PROGRAM S03_LidChecking
VAR
	//工站
	station					: REFERENCE TO FB_Station:=fbstation[3];
	//气缸
	fbHOZAdjustCyl_1	:REFERENCE TO FB_Cylinder:=fbCylinder[12];	//	上层水平调整气缸1（小）
	fbHOZAdjustCyl_2	:REFERENCE TO FB_Cylinder:=fbCylinder[13];	//	上层水平调整气缸2（小）
	fbHOZAdjustCyl_3	:REFERENCE TO FB_Cylinder:=fbCylinder[14];	//	下层水平调整气缸1（小）
	fbHOZAdjustCyl_4	:REFERENCE TO FB_Cylinder:=fbCylinder[15];	//	下层水平调整气缸2（小）
	fbHOZAdjustCyl_5	:REFERENCE TO FB_Cylinder:=fbCylinder[16];	//	上层水平调整气缸1（大）
	fbHOZAdjustCyl_6	:REFERENCE TO FB_Cylinder:=fbCylinder[17];	//	上层水平调整气缸2（大）
	fbHOZAdjustCyl_7	:REFERENCE TO FB_Cylinder:=fbCylinder[18];	//	下层水平调整气缸1（大）
	fbHOZAdjustCyl_8	:REFERENCE TO FB_Cylinder:=fbCylinder[19];	//	下层水平调整气缸2（大）
	//伺服
	fbXAxisMove	 :REFERENCE TO FB_Axis:=fbAxis[6];	//	相机检测工位X轴伺服
	fbYAxisMove	 :REFERENCE TO FB_Axis:=fbAxis[7];	//	相机检测工位Y轴伺服
	fbZAxisMove	 :REFERENCE TO FB_Axis:=fbAxis[8];	//	相机检测工位Z轴伺服
	//相机

	
		//延时
		arTonDelay :ARRAY[1..20] OF TON;
	//返回值
		UdiReturnValue :ARRAY[1..20] OF UDINT;
	//本地过程数据
	arProcessDataStation : ARRAY [1..5] OF DUT_MainlineFixture;
	
	i,j: INT;
	
	// 循环计数
	bCounter: BYTE;
	// 临时变量
	_FirstCycle:ARRAY[1..10] OF BOOL;
	them: INT;
	// X轴伺服循环次数
	bXCounter: BYTE;
	// Y轴伺服循环次数
	bYCounter: BYTE;
	// 结束时循环次数
	bEndCounter: INT;
	//相机检测工位检测结果
	arCameraResult:ARRAY[1..5,1..4,1..12] OF INT;
	//过程记录
	tsModuleProcess:ARRAY[1..gc_ModuleProNo] OF DUT_Process;
	xClearModuleProcessDone:BOOL;
	bClearProcessStep	:BYTE;
END_VAR

A_Input();
Alarm();
Delay();
FlowAuto();
FlowInit();
General();
ILC();
TipAuto();
TipManual();
Z_Output();

ACTION A_Input:
//气缸
fbHOZAdjustCyl_1.xWP_Sensor	:=	IxS03HOZAdjustCyl_1WP	;
fbHOZAdjustCyl_1.xHP_Sensor	:=	IxS03HOZAdjustCyl_1HP	;
fbHOZAdjustCyl_2.xWP_Sensor	:=	IxS03HOZAdjustCyl_2WP	;
fbHOZAdjustCyl_2.xHP_Sensor	:=	IxS03HOZAdjustCyl_2HP	;
fbHOZAdjustCyl_3.xWP_Sensor	:=	IxS03HOZAdjustCyl_3WP	;
fbHOZAdjustCyl_3.xHP_Sensor	:=	IxS03HOZAdjustCyl_3HP	;
fbHOZAdjustCyl_4.xWP_Sensor	:=	IxS03HOZAdjustCyl_4WP	;
fbHOZAdjustCyl_4.xHP_Sensor	:=	IxS03HOZAdjustCyl_4HP	;
fbHOZAdjustCyl_5.xWP_Sensor	:=	IxS03HOZAdjustCyl_5WP	;
fbHOZAdjustCyl_5.xHP_Sensor	:=	IxS03HOZAdjustCyl_5HP	;
fbHOZAdjustCyl_6.xWP_Sensor	:=	IxS03HOZAdjustCyl_6WP	;
fbHOZAdjustCyl_6.xHP_Sensor	:=	IxS03HOZAdjustCyl_6HP	;
fbHOZAdjustCyl_7.xWP_Sensor	:=	IxS03HOZAdjustCyl_7WP	;
fbHOZAdjustCyl_7.xHP_Sensor	:=	IxS03HOZAdjustCyl_7HP	;
fbHOZAdjustCyl_8.xWP_Sensor	:=	IxS03HOZAdjustCyl_8WP	;
fbHOZAdjustCyl_8.xHP_Sensor	:=	IxS03HOZAdjustCyl_8HP	;
END_ACTION

ACTION Alarm:
station.adwAlarm[1].00	:=	station.xInitTimeout	;//	S03 初始化超时
station.adwAlarm[1].01	:=	fbHOZAdjustCyl_1.xHP_Off 	;//	S03上层水平调整气缸1(小)原点未到位
station.adwAlarm[1].02	:=	fbHOZAdjustCyl_1.xWP_Off 	;//	S03上层水平调整气缸1(小)动点未到位
station.adwAlarm[1].03	:=	fbHOZAdjustCyl_2.xHP_Off	;//	S03上层水平调整气缸2(小)原点未到位
station.adwAlarm[1].04	:=	fbHOZAdjustCyl_2.xWP_Off	;//	S03上层水平调整气缸2(小)动点未到位
station.adwAlarm[1].05	:=	fbHOZAdjustCyl_3.xHP_Off	;//	S03下层水平调整气缸1(小)原点未到位
station.adwAlarm[1].06	:=	fbHOZAdjustCyl_3.xWP_Off	;//	S03下层水平调整气缸1(小)动点未到位
station.adwAlarm[1].07	:=	fbHOZAdjustCyl_4.xHP_Off	;//	S03下层水平调整气缸2(小)原点未到位
station.adwAlarm[1].08	:=	fbHOZAdjustCyl_4.xWP_Off	;//	S03下层水平调整气缸2(小)动点未到位
station.adwAlarm[1].09	:=	fbHOZAdjustCyl_5.xHP_Off	;//	S03上层水平调整气缸1(大)原点未到位
station.adwAlarm[1].10	:=	fbHOZAdjustCyl_5.xWP_Off	;//	S03上层水平调整气缸1(大)动点未到位
station.adwAlarm[1].11	:=	fbHOZAdjustCyl_6.xHP_Off	;//	S03上层水平调整气缸2(大)原点未到位
station.adwAlarm[1].12	:=	fbHOZAdjustCyl_6.xWP_Off	;//	S03上层水平调整气缸2(大)动点未到位
station.adwAlarm[1].13	:=	fbHOZAdjustCyl_7.xHP_Off	;//	S03下层水平调整气缸1(大)原点未到位
station.adwAlarm[1].14	:=	fbHOZAdjustCyl_7.xWP_Off	;//	S03下层水平调整气缸1(大)动点未到位
station.adwAlarm[1].15	:=	fbHOZAdjustCyl_8.xHP_Off	;//	S03下层水平调整气缸2(大)原点未到位
station.adwAlarm[1].16	:=	fbHOZAdjustCyl_8.xWP_Off	;//	S03下层水平调整气缸2(大)动点未到位
station.adwAlarm[1].17	:=	fbXAxisMove.xError	;//	S03液位检测X轴伺服报错
station.adwAlarm[1].18	:=	fbXAxisMove.xNotPowerOn	;//	S03液位检测X轴伺服未使能
station.adwAlarm[1].19	:=	fbXAxisMove.xMoveTimeout	;//	S03液位检测X轴伺服移动超时
station.adwAlarm[1].20	:=	fbYAxisMove.xError	;//	S03液位检测Y轴伺服报错
station.adwAlarm[1].21	:=	fbYAxisMove.xNotPowerOn	;//	S03液位检测Y轴伺服未使能
station.adwAlarm[1].22	:=	fbYAxisMove.xMoveTimeout	;//	S03液位检测Y轴伺服移动超时
station.adwAlarm[1].23	:=	fbZAxisMove.xError	;//	S03液位检测Z轴伺服报错
station.adwAlarm[1].24	:=	fbZAxisMove.xNotPowerOn	;//	S03液位检测Z轴伺服未使能
station.adwAlarm[1].25	:=	fbZAxisMove.xMoveTimeout	;//	S03液位检测Z轴伺服移动超时
END_ACTION

ACTION Delay:
(*arTonDelay[01](IN:= , PT:=T#0.1S , Q=> , ET=> );*)//TipAuto使用
arTonDelay[02](IN:=  , PT:=T#1S , Q=> , ET=> );
arTonDelay[03](IN:=   , PT:=T#1S , Q=> , ET=> );
arTonDelay[04](IN:= , PT:=T#0.1S , Q=> , ET=> );
arTonDelay[05](IN:= , PT:=T#0.1S , Q=> , ET=> );
arTonDelay[06](IN:= , PT:=T#0.1S , Q=> , ET=> );
arTonDelay[07](IN:= , PT:=T#0.1S , Q=> , ET=> );
arTonDelay[08](IN:= , PT:=T#0.1S , Q=> , ET=> );
arTonDelay[09](IN:= , PT:=T#0.1S , Q=> , ET=> );
END_ACTION

ACTION FlowAuto:

//-----------------------------------------初始化是否完成判断----------------------------------------------
IF NOT station.xInitDone 
THEN
 	station.iStepAuto:=0;
 	station.xDone:=FALSE;
	station.xRunningOffProhibit := FALSE ;//运行中信号Off禁止
ELSIF station.xRunning  OR (tsModuleProcess[bXCounter+1].xProcessStarted AND NOT tsModuleProcess[bXCounter+1].xProcessCompleted)
THEN
//-----------------------------------------动作步骤--------------------------------------------------------
CASE station.iStepAuto OF	  
	0: //----Home Step，等待启动----
		IF station.xDisabled 
			AND station.xCanRun 
			AND NOT fbMachine[1].xStopped 
			AND NOT station.xSingleRunning 
		THEN
			station.xDone:=TRUE;
		END_IF
		
		IF  station.xSingleRunning 
			OR station.xCanRun 
			AND NOT station.xDone 
			AND NOT station.xDisabled 
			AND NOT fbMachine[1].xStopped
		THEN
			station.xCycleEnable:=TRUE;
			station.xDone:= FALSE;  
			station.iStepAuto:= 5;
		END_IF		
	 5://复位数据
			IF  station.xSingleRunning THEN
				 FOR i:=1 TO gc_ModuleProNo BY 1 DO
						 MEMSET(ADR(tsModuleProcess[i]),0,SIZEOF(tsModuleProcess[i]));
				 END_FOR
			END_IF	
			station.iStepAuto:= 10;
	 10: //判断产品是否到该工位
		IF  station.xSingleRunning THEN
			station.iStepAuto:= 11;
		ELSIF fbMachine[1].xTryRun THEN
			IF NOT _FirstCycle[6] THEN
					bCounter:=1;
					bEndCounter:=0;
				_FirstCycle[6]:=TRUE;
			END_IF
			station.iStepAuto:= 11;
		ELSE
			IF   	 NOT  arMainlineFixtureData[arCurFixtureNumStation[5]].xMaterialOnOff AND
					 NOT arMainlineFixtureData[arCurFixtureNumStation[6]].xMaterialOnOff  AND 
					 NOT arMainlineFixtureData[arCurFixtureNumStation[7]].xMaterialOnOff AND 
					NOT	arMainlineFixtureData[arCurFixtureNumStation[8]].xMaterialOnOff AND
					NOT arMainlineFixtureData[arCurFixtureNumStation[9]].xMaterialOnOff  THEN
							bCounter:=0;
							bEndCounter :=0;
							_FirstCycle[1]:=FALSE;
							_FirstCycle[2]:=FALSE;
							_FirstCycle[6]:=FALSE;
							station.iStepAuto:= 999;
						
			ELSIF	 arMainlineFixtureData[arCurFixtureNumStation[5]].xMaterialOnOff AND    
				    arMainlineFixtureData[arCurFixtureNumStation[6]].xMaterialOnOff (* AND 
				NOT arMainlineFixtureData[arCurFixtureNumStation[7]].xMaterialOnOff AND 
				NOT	arMainlineFixtureData[arCurFixtureNumStation[8]].xMaterialOnOff AND
				NOT arMainlineFixtureData[arCurFixtureNumStation[9]].xMaterialOnOff*)  THEN
					IF  NOT _FirstCycle[1] THEN
							bCounter:=1;
							bEndCounter :=0;
							_FirstCycle[1]:=TRUE;
					END_IF
					station.iStepAuto:= 11;
			ELSIF   NOT arMainlineFixtureData[arCurFixtureNumStation[5]].xMaterialOnOff AND    
				    NOT arMainlineFixtureData[arCurFixtureNumStation[6]].xMaterialOnOff  AND 
						arMainlineFixtureData[arCurFixtureNumStation[7]].xMaterialOnOff AND 
						arMainlineFixtureData[arCurFixtureNumStation[8]].xMaterialOnOff AND
						arMainlineFixtureData[arCurFixtureNumStation[9]].xMaterialOnOff  THEN
					IF  NOT _FirstCycle[2] THEN
							bEndCounter:=1;
							bCounter:=0;
							_FirstCycle[2]:=TRUE;
					END_IF
					station.iStepAuto:= 11;
			END_IF
		END_IF
	11://手动NOK按钮
			IF   arManualNOKHmiButton[3]  AND NOT station.xSingleRunning THEN
				station.iStepAuto:= 280;
			ELSE	
				station.iStepAuto:= 20;
			END_IF
			
	20:////Restore_after_Estop_Process1 上载数据流程
			IF   station.xSingleRunning OR  fbMachine[1].xTryRun THEN
				    station.iStepAuto :=40;
			ELSIF tsModuleProcess[1].xProcessNotStarted AND NOT  tsModuleProcess[1].xProcessStarted THEN
					station.iStepAuto :=21; (*process not started*)
			ELSIF  tsModuleProcess[1].xProcessStarted AND NOT  tsModuleProcess[1].xProcessCompleted THEN
				 station.iStepAuto := 21;(*process started*)
			ELSIF  tsModuleProcess[1].xProcessCompleted AND NOT tsModuleProcess[1].xQDataCompleted  THEN
					station.iStepAuto := 40 ;(*process completed*)
			ELSIF tsModuleProcess[1].xQDataCompleted THEN
					station.iStepAuto :=40;(*Qdata completed *)
			ELSE
					station.iStepAuto :=21; 
			END_IF	
	21://
				tsModuleProcess[1].xProcessNotStarted:=TRUE;
				station.iStepAuto:= 30;
	30://上载产品数据
			tsModuleProcess[1].xProcessStarted	:=TRUE;
			IF  bCounter =1 OR bCounter =2 OR bCounter=3 THEN
				MEMCPY(ADR(arProcessDataStation[1]),ADR(arMainlineFixtureData[arCurFixtureNumStation[5]]),SIZEOF(arMainlineFixtureData[arCurFixtureNumStation[5]]));
				MEMCPY(ADR(arProcessDataStation[2]),ADR(arMainlineFixtureData[arCurFixtureNumStation[6]]),SIZEOF(arMainlineFixtureData[arCurFixtureNumStation[6]]))	;
			END_IF
			IF bCounter =2 OR bCounter =3 OR bEndCounter =1 THEN
				MEMCPY(ADR(arProcessDataStation[3]),ADR(arMainlineFixtureData[arCurFixtureNumStation[7]]),SIZEOF(arMainlineFixtureData[arCurFixtureNumStation[7]]));
				MEMCPY(ADR(arProcessDataStation[4]),ADR(arMainlineFixtureData[arCurFixtureNumStation[8]]),SIZEOF(arMainlineFixtureData[arCurFixtureNumStation[8]]))	;
			END_IF
			IF bCounter =3 OR bEndCounter =2 THEN
				MEMCPY(ADR(arProcessDataStation[5]),ADR(arMainlineFixtureData[arCurFixtureNumStation[9]]),SIZEOF(arMainlineFixtureData[arCurFixtureNumStation[9]]))	;
			END_IF
			tsModuleProcess[1].xProcessCompleted:=TRUE;
			station.iStepAuto:= 40;
	/////产品流程开始	
		40://设定X轴循环为1，总次数2
				 bXCounter:=1;
				station.iStepAuto:= 50;		
		50:////Restore_after_Estop_Process2/3 X轴位置1/2拍照流程
			 IF  station.xSingleRunning OR fbMachine[1].xTryRun THEN
					 station.iStepAuto :=70; 
			 ELSIF tsModuleProcess[bXCounter+1].xProcessNotStarted AND NOT  tsModuleProcess[bXCounter+1].xProcessStarted THEN
					 station.iStepAuto :=70; (*process not started*)
			 ELSIF  tsModuleProcess[bXCounter+1].xProcessStarted AND NOT  tsModuleProcess[bXCounter+1].xProcessCompleted THEN
					station.iStepAuto := 70;(*process started*)
			 ELSIF  tsModuleProcess[bXCounter+1].xProcessCompleted AND NOT tsModuleProcess[bXCounter+1].xQDataCompleted  THEN
					 station.iStepAuto :=200;(*process completed*)
			 ELSIF tsModuleProcess[bXCounter+1].xQDataCompleted THEN
					 station.iStepAuto :=200;(*Qdata completed *)
			 ELSE
					 station.iStepAuto :=70; 
			 END_IF	
		70://流程未开始
				tsModuleProcess[bXCounter+1].xProcessNotStarted :=TRUE;
				station.iStepAuto :=80; 
		80://水平调整气缸伸出		
			IF   bCounter =1 THEN
					IF  iBoxChoose =1 THEN
						(*上层水平调整气缸*)
						fbHOZAdjustCyl_1.xAuto :=TRUE;
						fbHOZAdjustCyl_2.xAuto :=TRUE;
						IF  fbHOZAdjustCyl_1.xWP_Delay AND fbHOZAdjustCyl_2.xWP_Delay  THEN
								station.iStepAuto:= 90;
						END_IF
					ELSIF  iBoxChoose= 2 THEN
						(*下层水平调整气缸*)
						fbHOZAdjustCyl_3.xAuto :=TRUE;
						fbHOZAdjustCyl_4.xAuto :=TRUE;
						IF  fbHOZAdjustCyl_3.xWP_Delay AND fbHOZAdjustCyl_4.xWP_Delay  THEN
								station.iStepAuto:= 90;
						END_IF
					END_IF
			ELSIF  bCounter =2 OR  bCounter =3 OR bEndCounter =1 OR bEndCounter =2 THEN
					IF  iBoxChoose =1 THEN
						(*上层水平调整气缸*)
						fbHOZAdjustCyl_5.xAuto :=TRUE;
						fbHOZAdjustCyl_6.xAuto :=TRUE;
						IF  fbHOZAdjustCyl_5.xWP_Delay AND fbHOZAdjustCyl_6.xWP_Delay  THEN
								station.iStepAuto:= 90;
						END_IF
					ELSIF  iBoxChoose= 2 THEN
						(*下层水平调整气缸*)
						fbHOZAdjustCyl_7.xAuto :=TRUE;
						fbHOZAdjustCyl_8.xAuto :=TRUE;
						IF  fbHOZAdjustCyl_7.xWP_Delay AND fbHOZAdjustCyl_8.xWP_Delay  THEN
								station.iStepAuto:= 90;
						END_IF
					END_IF
			END_IF
		90://Z轴下降
			fbZAxisMove.xMoveAuto[2]:=TRUE;
			IF  fbXAxisMove.xMoveInPos[2] THEN
				station.iStepAuto:= 95;
			END_IF			 
		95://X轴移动到拍照位置1/2
				fbXAxisMove.xMoveAuto[bXCounter+1]:=TRUE;
				IF  fbXAxisMove.xMoveInPos[bXCounter+1] THEN
					station.iStepAuto:= 100;
				END_IF
		100://设定Y轴循环开始 总次数为3
				 bYCounter:=1;
				station.iStepAuto:= 110;	
		110://Y轴移动到位置1/2/3	
				fbYAxisMove.xMoveAuto[bYCounter+1]:=TRUE;
				IF  fbYAxisMove.xMoveInPos[bYCounter+1] THEN
					station.iStepAuto:= 120;
				END_IF
		120://屏蔽拍照
			IF axBypassSignal[3] OR  fbMachine[1].xTryRun THEN
 					station.iStepAuto:= 150;	
			ELSE
					station.iStepAuto:= 140;		
			END_IF
		140://触发拍照
			(*开始循环*)
			tsModuleProcess[bXCounter+1].xProcessStarted :=TRUE;
			IF   bCounter =1  (*17.18位置有产品*)  THEN
					IF  bXCounter =1 THEN
							FOR i:=2 TO  9 BY 1 DO
								fbCamera[i].xlTrigger:=TRUE;
							END_FOR
					ELSIF bXCounter =2 THEN
							FOR i:=2 TO  5 BY 1 DO
								fbCamera[i].xlTrigger:=TRUE;
							END_FOR
					END_IF
			ELSIF  bCounter=2  THEN
					IF  bXCounter =1 THEN
								FOR i:=2 TO 17 BY 1 DO
									fbCamera[i].xlTrigger:=TRUE;
								END_FOR
					ELSIF   bXCounter =2 THEN
								FOR i:=2 TO 13 BY 1 DO
									fbCamera[i].xlTrigger:=TRUE;
								END_FOR	
					END_IF
			ELSIF   bCounter=3 THEN
					FOR i:=2 TO 17 BY 1 DO
						fbCamera[i].xlTrigger:=TRUE;
					END_FOR
			END_IF
			(*结束循环*)
			IF   bEndCounter =1 (*17.18位置无产品*)  THEN
					IF  bXCounter =1 THEN
								FOR i:=6 TO  17 BY 1 DO
									fbCamera[i].xlTrigger:=TRUE;
								END_FOR
					ELSIF bXCounter =2 THEN
								FOR i:=2 TO  17 BY 1 DO
									fbCamera[i].xlTrigger:=TRUE;
								END_FOR
					END_IF
			ELSIF  bEndCounter =2 THEN
					IF bXCounter =2 THEN
							FOR i:=14 TO  17 BY 1 DO
									fbCamera[i].xlTrigger:=TRUE;
							END_FOR	
					END_IF
			END_IF
			FOR i:=2 TO 17 BY 1 DO
				IF  fbCamera[i].xQBusy  THEN
					fbCamera[i].xlTrigger:=FALSE;
					station.iStepAuto:=150;
				END_IF
			END_FOR
		150://检查相机完成信号并储存
		(*开始循环*)
			 IF   bCounter =1 (*17.18位置有产品*)  THEN	
				  	IF  bXCounter =1 THEN
							IF   axBypassSignal[3] OR  fbMachine[1].xTryRun THEN
								
											arCameraResult[1,3,bYCounter]:=1;	
											arCameraResult[1,3,6+bYCounter]:=1;	
											arCameraResult[1,1,3+bYCounter]:=1;
											arCameraResult[1,1,9+bYCounter]:=1;
											arCameraResult[2,4,bYCounter]:=1;
											arCameraResult[2,4,6+bYCounter]:=1;
											arCameraResult[2,2,3+bYCounter]:=1;
											arCameraResult[2,2,9+bYCounter]:=1;	
											station.iStepAuto:=160;
							ELSE
								FOR i:=1 TO  8 BY 1 DO
										IF  fbCamera[i].xQBusy THEN	
												EXIT;
										ELSE
												IF  i =1 THEN
													arCameraResult[1,3,bYCounter]:=sCamera_To_Plc.iS03Result[i];	
												ELSIF i =2 THEN
													arCameraResult[1,3,6+bYCounter]:=sCamera_To_Plc.iS03Result[i];	
												ELSIF i =3 THEN
													arCameraResult[1,1,3+bYCounter]:=sCamera_To_Plc.iS03Result[i];
												ELSIF i =4 THEN
													arCameraResult[1,1,9+bYCounter]:=sCamera_To_Plc.iS03Result[i];
												ELSIF i =5 THEN
													arCameraResult[2,4,bYCounter]:=sCamera_To_Plc.iS03Result[i];
												ELSIF i =6 THEN
													arCameraResult[2,4,6+bYCounter]:=sCamera_To_Plc.iS03Result[i];
												ELSIF i =7 THEN
													arCameraResult[2,2,3+bYCounter]:=sCamera_To_Plc.iS03Result[i];
												ELSIF i =8 THEN
													arCameraResult[2,2,9+bYCounter]:=sCamera_To_Plc.iS03Result[i];	
												END_IF	
										END_IF
										IF   i =8 THEN
											station.iStepAuto:=160;
										END_IF
								END_FOR
							END_IF
				
				 	ELSIF   bXCounter =2 THEN
							IF   axBypassSignal[3] OR  fbMachine[1].xTryRun THEN
											arCameraResult[2,3,bYCounter]:=1;	
											arCameraResult[2,3,6+bYCounter]:=1;	
											arCameraResult[2,1,3+bYCounter]:=1;
											arCameraResult[2,1,9+bYCounter]:=1;
											station.iStepAuto:=160;
							ELSE
								FOR i:=1 TO 4 BY 1	DO
										IF  fbCamera[i].xQBusy THEN	
											EXIT;
										ELSE
											IF  i =1 THEN
												arCameraResult[2,3,bYCounter]:=sCamera_To_Plc.iS03Result[i];	
											ELSIF i =2 THEN
												arCameraResult[2,3,6+bYCounter]:=sCamera_To_Plc.iS03Result[i];	
											ELSIF i =3 THEN
												arCameraResult[2,1,3+bYCounter]:=sCamera_To_Plc.iS03Result[i];
											ELSIF i =4 THEN
												arCameraResult[2,1,9+bYCounter]:=sCamera_To_Plc.iS03Result[i];
											END_IF
										END_IF	
										IF   i =8 THEN
											station.iStepAuto:=160;
										END_IF
								END_FOR
							END_IF
							
					END_IF		
			ELSIF  bCounter=2 THEN
					IF bXCounter =1 THEN
							IF   axBypassSignal[3] OR  fbMachine[1].xTryRun THEN
									
												arCameraResult[1,3,bYCounter]:=1;	
												arCameraResult[1,3,6+bYCounter]:=1;	
												arCameraResult[1,1,3+bYCounter]:=1;
												arCameraResult[1,1,9+bYCounter]:=1;
												arCameraResult[2,4,bYCounter]:=1;
												arCameraResult[2,4,6+bYCounter]:=1;
												arCameraResult[2,2,3+bYCounter]:=1;
												arCameraResult[2,2,9+bYCounter]:=1;	
												arCameraResult[3,3,3+bYCounter]:=1;	
												arCameraResult[3,3,9+bYCounter]:=1;	
												arCameraResult[3,1,bYCounter]:= 1;
												arCameraResult[3,1,6+bYCounter]:=1;
												arCameraResult[4,4,3+bYCounter]:=1;
												arCameraResult[4,4,9+bYCounter]:=1;
												arCameraResult[4,2,3+bYCounter]:=1;
												arCameraResult[4,2,6+bYCounter]:=1;	
												station.iStepAuto:=160;
							ELSE
								FOR i:=1 TO  16 BY 1 DO
									IF  fbCamera[i].xQBusy THEN	
											EXIT;
									ELSE
											IF  i =1 THEN
												arCameraResult[1,3,bYCounter]:=sCamera_To_Plc.iS03Result[i];	
											ELSIF i =2 THEN
												arCameraResult[1,3,6+bYCounter]:=sCamera_To_Plc.iS03Result[i];	
											ELSIF i =3 THEN
												arCameraResult[1,1,3+bYCounter]:=sCamera_To_Plc.iS03Result[i];
											ELSIF i =4 THEN
												arCameraResult[1,1,9+bYCounter]:=sCamera_To_Plc.iS03Result[i];
											ELSIF i =5 THEN
												arCameraResult[2,4,bYCounter]:=sCamera_To_Plc.iS03Result[i];
											ELSIF i =6 THEN
												arCameraResult[2,4,6+bYCounter]:=sCamera_To_Plc.iS03Result[i];
											ELSIF i =7 THEN
												arCameraResult[2,2,3+bYCounter]:=sCamera_To_Plc.iS03Result[i];
											ELSIF i =8 THEN
												arCameraResult[2,2,9+bYCounter]:=sCamera_To_Plc.iS03Result[i];	
											ELSIF i =9 THEN
												arCameraResult[3,3,3+bYCounter]:=sCamera_To_Plc.iS03Result[i];	
											ELSIF i =10 THEN
												arCameraResult[3,3,9+bYCounter]:=sCamera_To_Plc.iS03Result[i];	
											ELSIF i =11 THEN
												arCameraResult[3,1,bYCounter]:=sCamera_To_Plc.iS03Result[i];
											ELSIF i =12 THEN
												arCameraResult[3,1,6+bYCounter]:=sCamera_To_Plc.iS03Result[i];
											ELSIF i =13 THEN
												arCameraResult[4,4,3+bYCounter]:=sCamera_To_Plc.iS03Result[i];
											ELSIF i =14 THEN
												arCameraResult[4,4,9+bYCounter]:=sCamera_To_Plc.iS03Result[i];
											ELSIF i =15 THEN
												arCameraResult[4,2,3+bYCounter]:=sCamera_To_Plc.iS03Result[i];
											ELSIF i =16 THEN
												arCameraResult[4,2,6+bYCounter]:=sCamera_To_Plc.iS03Result[i];	
											END_IF	
									END_IF	
									IF   i =16 THEN
											station.iStepAuto:=160;
									END_IF
								END_FOR	
							END_IF
							
					ELSIF bXCounter =2 THEN
							IF   axBypassSignal[3] OR  fbMachine[1].xTryRun THEN
											arCameraResult[2,3,bYCounter]:=1;	
											arCameraResult[2,3,6+bYCounter]:=1;	
											arCameraResult[2,1,3+bYCounter]:=1;
											arCameraResult[2,1,9+bYCounter]:=1;
											arCameraResult[3,4,bYCounter]:=1;
											arCameraResult[3,4,6+bYCounter]:=1;
											arCameraResult[3,2,3+bYCounter]:=1;
											arCameraResult[3,2,9+bYCounter]:=1;	
											arCameraResult[4,3,3+bYCounter]:=1;	
											arCameraResult[4,3,9+bYCounter]:=1;	
											arCameraResult[4,1,bYCounter]:=1;
											arCameraResult[4,1,6+bYCounter]:=1;
											station.iStepAuto:=160;
							ELSE
								FOR i:=1 TO  12 BY 1 DO
									IF  fbCamera[i].xQBusy THEN	
											EXIT;
									ELSE
											IF  i =1 THEN
												arCameraResult[2,3,bYCounter]:=sCamera_To_Plc.iS03Result[i];	
											ELSIF i =2 THEN       
												arCameraResult[2,3,6+bYCounter]:=sCamera_To_Plc.iS03Result[i];	
											ELSIF i =3 THEN      
												arCameraResult[2,1,3+bYCounter]:=sCamera_To_Plc.iS03Result[i];
											ELSIF i =4 THEN      
												arCameraResult[2,1,9+bYCounter]:=sCamera_To_Plc.iS03Result[i];
											ELSIF i =5 THEN      
												arCameraResult[3,4,bYCounter]:=sCamera_To_Plc.iS03Result[i];
											ELSIF i =6 THEN     
												arCameraResult[3,4,6+bYCounter]:=sCamera_To_Plc.iS03Result[i];
											ELSIF i =7 THEN      
												arCameraResult[3,2,3+bYCounter]:=sCamera_To_Plc.iS03Result[i];
											ELSIF i =8 THEN      
												arCameraResult[3,2,9+bYCounter]:=sCamera_To_Plc.iS03Result[i];	
											ELSIF i =9 THEN      
												arCameraResult[4,3,3+bYCounter]:=sCamera_To_Plc.iS03Result[i];	
											ELSIF i =10 THEN     
												arCameraResult[4,3,9+bYCounter]:=sCamera_To_Plc.iS03Result[i];	
											ELSIF i =11 THEN      
												arCameraResult[4,1,bYCounter]:=sCamera_To_Plc.iS03Result[i];
											ELSIF i =12 THEN      
												arCameraResult[4,1,6+bYCounter]:=sCamera_To_Plc.iS03Result[i];
											END_IF	
									END_IF
									IF   i =12 THEN
										station.iStepAuto:=160;
									END_IF	
								END_FOR	
							END_IF
					END_IF
				
			ELSIF  bCounter =3 THEN
					IF bXCounter =1 THEN
							IF   axBypassSignal[3] OR  fbMachine[1].xTryRun THEN
								
											arCameraResult[1,3,bYCounter]:=	1;	
											arCameraResult[1,3,6+bYCounter]:=1;	
											arCameraResult[1,1,3+bYCounter]:=1;
											arCameraResult[1,1,9+bYCounter]:=1;
											arCameraResult[2,4,bYCounter]:=1;
											arCameraResult[2,4,6+bYCounter]:=1;
											arCameraResult[2,2,3+bYCounter]:=1;
											arCameraResult[2,2,9+bYCounter]:=1;	
											arCameraResult[3,3,3+bYCounter]:=1;	
											arCameraResult[3,3,9+bYCounter]:=1;	
											arCameraResult[3,1,bYCounter]:=1;
											arCameraResult[3,1,6+bYCounter]:=1;
											arCameraResult[4,4,3+bYCounter]:=1;
											arCameraResult[4,4,9+bYCounter]:=1;
											arCameraResult[4,2,3+bYCounter]:=1;
											arCameraResult[4,2,6+bYCounter]:=1;	
											station.iStepAuto:=160;
							ELSE
								FOR i:=1 TO  16 BY 1 DO
										IF  fbCamera[i].xQBusy THEN	
												EXIT;
										ELSE
												IF  i =1 THEN
													arCameraResult[1,3,bYCounter]:=sCamera_To_Plc.iS03Result[i];	
												ELSIF i =2 THEN   
													arCameraResult[1,3,6+bYCounter]:=sCamera_To_Plc.iS03Result[i];	
												ELSIF i =3 THEN    
													arCameraResult[1,1,3+bYCounter]:=sCamera_To_Plc.iS03Result[i];
												ELSIF i =4 THEN    
													arCameraResult[1,1,9+bYCounter]:=sCamera_To_Plc.iS03Result[i];
												ELSIF i =5 THEN     
													arCameraResult[2,4,bYCounter]:=sCamera_To_Plc.iS03Result[i];
												ELSIF i =6 THEN    
													arCameraResult[2,4,6+bYCounter]:=sCamera_To_Plc.iS03Result[i];
												ELSIF i =7 THEN     
													arCameraResult[2,2,3+bYCounter]:=sCamera_To_Plc.iS03Result[i];
												ELSIF i =8 THEN     
													arCameraResult[2,2,9+bYCounter]:=sCamera_To_Plc.iS03Result[i];	
												ELSIF i =9 THEN     
													arCameraResult[3,3,3+bYCounter]:=sCamera_To_Plc.iS03Result[i];	
												ELSIF i =10 THEN    
													arCameraResult[3,3,9+bYCounter]:=sCamera_To_Plc.iS03Result[i];	
												ELSIF i =11 THEN    
													arCameraResult[3,1,bYCounter]:=sCamera_To_Plc.iS03Result[i];
												ELSIF i =12 THEN    
													arCameraResult[3,1,6+bYCounter]:=sCamera_To_Plc.iS03Result[i];
												ELSIF i =13 THEN    
													arCameraResult[4,4,3+bYCounter]:=sCamera_To_Plc.iS03Result[i];
												ELSIF i =14 THEN    
													arCameraResult[4,4,9+bYCounter]:=sCamera_To_Plc.iS03Result[i];
												ELSIF i =15 THEN    
													arCameraResult[4,2,3+bYCounter]:=sCamera_To_Plc.iS03Result[i];
												ELSIF i =16 THEN   
													arCameraResult[4,2,6+bYCounter]:=sCamera_To_Plc.iS03Result[i];	
												END_IF	
										END_IF	
										IF  i =16 THEN 
											station.iStepAuto:=160;
										END_IF
								END_FOR	
							END_IF
					ELSIF bXCounter =2 THEN
							IF   axBypassSignal[3] OR  fbMachine[1].xTryRun THEN
								
												arCameraResult[2,3,bYCounter]:=1;	
											arCameraResult[2,3,6+bYCounter]:=1;	
											arCameraResult[2,1,3+bYCounter]:=1;
											arCameraResult[2,1,9+bYCounter]:=1;
											arCameraResult[3,4,bYCounter]:=1;
											arCameraResult[3,4,6+bYCounter]:=1;
											arCameraResult[3,2,3+bYCounter]:=1;
											arCameraResult[3,2,9+bYCounter]:=1;	
											arCameraResult[4,3,3+bYCounter]:=1;	
											arCameraResult[4,3,9+bYCounter]:=1;	
											arCameraResult[4,1,bYCounter]:=1;
											arCameraResult[4,1,6+bYCounter]:=1;
											arCameraResult[5,4,3+bYCounter]:=1;
											arCameraResult[5,4,9+bYCounter]:=1;
											arCameraResult[5,2,3+bYCounter]:=1;
											arCameraResult[5,2,6+bYCounter]:=1;	
											station.iStepAuto:=160;
							ELSE
								FOR i:=1 TO  12 BY 1 DO
									IF fbCamera[i].xQBusy THEN	
											EXIT;
									ELSE
											IF  i =1 THEN
												arCameraResult[2,3,bYCounter]:=sCamera_To_Plc.iS03Result[i];	
											ELSIF i =2 THEN   
												arCameraResult[2,3,6+bYCounter]:=sCamera_To_Plc.iS03Result[i];	
											ELSIF i =3 THEN    
												arCameraResult[2,1,3+bYCounter]:=sCamera_To_Plc.iS03Result[i];
											ELSIF i =4 THEN     
												arCameraResult[2,1,9+bYCounter]:=sCamera_To_Plc.iS03Result[i];
											ELSIF i =5 THEN     
												arCameraResult[3,4,bYCounter]:=sCamera_To_Plc.iS03Result[i];
											ELSIF i =6 THEN    
												arCameraResult[3,4,6+bYCounter]:=sCamera_To_Plc.iS03Result[i];
											ELSIF i =7 THEN   
												arCameraResult[3,2,3+bYCounter]:=sCamera_To_Plc.iS03Result[i];
											ELSIF i =8 THEN     
												arCameraResult[3,2,9+bYCounter]:=sCamera_To_Plc.iS03Result[i];	
											ELSIF i =9 THEN    
												arCameraResult[4,3,3+bYCounter]:=sCamera_To_Plc.iS03Result[i];	
											ELSIF i =10 THEN    
												arCameraResult[4,3,9+bYCounter]:=sCamera_To_Plc.iS03Result[i];	
											ELSIF i =11 THEN    
												arCameraResult[4,1,bYCounter]:=sCamera_To_Plc.iS03Result[i];
											ELSIF i =12 THEN    
												arCameraResult[4,1,6+bYCounter]:=sCamera_To_Plc.iS03Result[i];
											ELSIF i =13 THEN   
												arCameraResult[5,4,3+bYCounter]:=sCamera_To_Plc.iS03Result[i];
											ELSIF i =14 THEN    
												arCameraResult[5,4,9+bYCounter]:=sCamera_To_Plc.iS03Result[i];
											ELSIF i =15 THEN    
												arCameraResult[5,2,3+bYCounter]:=sCamera_To_Plc.iS03Result[i];
											ELSIF i =16 THEN   
												arCameraResult[5,2,6+bYCounter]:=sCamera_To_Plc.iS03Result[i];	
											END_IF	
									END_IF
									IF  i =12 THEN
										station.iStepAuto:=160;	
									END_IF
								END_FOR	
							END_IF
					END_IF
			END_IF
			
		(*结束循环*)
			 IF   bEndCounter =1 (*17.18位置无产品*)  THEN	
				  	IF  bXCounter =1 THEN
							IF   axBypassSignal[3] OR  fbMachine[1].xTryRun THEN
											arCameraResult[3,3,3+bYCounter]:=1;
											arCameraResult[3,3,9+bYCounter]:=1;
											arCameraResult[3,1,bYCounter]:=1;
											arCameraResult[3,1,3+bYCounter]:=1;                 
											arCameraResult[4,4,3+bYCounter]:=1;	
											arCameraResult[4,4,9+bYCounter]:=1;
											arCameraResult[4,2,bYCounter]:=1;
											arCameraResult[4,2,6+bYCounter]:=1;
											station.iStepAuto:=160;
							ELSE
								FOR i:=9 TO  16 BY 1 DO
									IF  fbCamera[i].xQBusy THEN	
											EXIT;
									ELSE
											IF i =9 THEN
												arCameraResult[3,3,3+bYCounter]:=sCamera_To_Plc.iS03Result[i];
											ELSIF i =10 THEN   
												arCameraResult[3,3,9+bYCounter]:=sCamera_To_Plc.iS03Result[i];
											ELSIF i =11 THEN   
												arCameraResult[3,1,bYCounter]:=sCamera_To_Plc.iS03Result[i];
											ELSIF i =12 THEN    
												arCameraResult[3,1,3+bYCounter]:=sCamera_To_Plc.iS03Result[i];                 
											ELSIF i =13 THEN   
												arCameraResult[4,4,3+bYCounter]:=sCamera_To_Plc.iS03Result[i];	
											ELSIF i =14 THEN    
												arCameraResult[4,4,9+bYCounter]:=sCamera_To_Plc.iS03Result[i];
											ELSIF i =15 THEN    
												arCameraResult[4,2,bYCounter]:=sCamera_To_Plc.iS03Result[i];
											ELSIF i =16 THEN   
												arCameraResult[4,2,6+bYCounter]:=sCamera_To_Plc.iS03Result[i];
											END_IF
									END_IF	
									IF  i =16 THEN
											station.iStepAuto:=160;	
									END_IF
								END_FOR	
							END_IF
							
				 	ELSIF   bXCounter =2 THEN
							IF   axBypassSignal[3] OR  fbMachine[1].xTryRun THEN
							
											arCameraResult[3,4,bYCounter]:=1;	
											arCameraResult[3,4,6+bYCounter]:=1;	
											arCameraResult[3,2,3+bYCounter]:=1;
											arCameraResult[3,2,9+bYCounter]:=1;
											arCameraResult[4,3,3+bYCounter]:=1;	
											arCameraResult[4,3,8+bYCounter]:=1;	
											arCameraResult[4,1,bYCounter]:=1;
											arCameraResult[4,1,6+bYCounter]:=1;		
											arCameraResult[5,4,3+bYCounter]:=1;	
											arCameraResult[5,4,9+bYCounter]:=1;	
											arCameraResult[5,2,bYCounter]:=1;
											arCameraResult[5,2,6+bYCounter]:=1;
											station.iStepAuto:=160;
							ELSE
								FOR i:=5 TO 16 BY 1	DO
										IF  fbCamera[i].xQBusy THEN	
											EXIT;
										ELSE
											IF  i =5 THEN
												arCameraResult[3,4,bYCounter]:=sCamera_To_Plc.iS03Result[i];	
											ELSIF i =6 THEN    
												arCameraResult[3,4,6+bYCounter]:=sCamera_To_Plc.iS03Result[i];	
											ELSIF i =7 THEN    
												arCameraResult[3,2,3+bYCounter]:=sCamera_To_Plc.iS03Result[i];
											ELSIF i =8 THEN    
												arCameraResult[3,2,9+bYCounter]:=sCamera_To_Plc.iS03Result[i];
											ELSIF  i =9 THEN    
												arCameraResult[4,3,3+bYCounter]:=sCamera_To_Plc.iS03Result[i];	
											ELSIF i =10 THEN    
												arCameraResult[4,3,8+bYCounter]:=sCamera_To_Plc.iS03Result[i];	
											ELSIF i =11 THEN    
												arCameraResult[4,1,bYCounter]:=sCamera_To_Plc.iS03Result[i];
											ELSIF i =12 THEN  
												arCameraResult[4,1,6+bYCounter]:=sCamera_To_Plc.iS03Result[i];		
											ELSIF  i =13 THEN 
												arCameraResult[5,4,3+bYCounter]:=sCamera_To_Plc.iS03Result[i];	
											ELSIF i =14 THEN   
												arCameraResult[5,4,9+bYCounter]:=sCamera_To_Plc.iS03Result[i];	
											ELSIF i =15 THEN   
												arCameraResult[5,2,bYCounter]:=sCamera_To_Plc.iS03Result[i];
											ELSIF i =16 THEN  
												arCameraResult[5,2,6+bYCounter]:=sCamera_To_Plc.iS03Result[i];
											END_IF
										END_IF
										IF i =16 THEN
											station.iStepAuto:=160;
										END_IF
								END_FOR
							END_IF
							
						END_IF		
			ELSIF  bEndCounter=2 THEN
					IF bXCounter =2 THEN
							IF   axBypassSignal[3] OR  fbMachine[1].xTryRun THEN
								
												arCameraResult[5,4,3+bYCounter]:=1;	
												arCameraResult[5,4,9+bYCounter]:=1;	
												arCameraResult[5,4,bYCounter]:=1;
												arCameraResult[5,4,6+bYCounter]:=1;
												station.iStepAuto:=160;
							ELSE
								FOR i:=13 TO  16 BY 1 DO
									IF  fbCamera[i].xQBusy THEN	
											EXIT;
									ELSE
											IF  i =13 THEN
												arCameraResult[5,4,3+bYCounter]:=sCamera_To_Plc.iS03Result[i];	
											ELSIF i =14 THEN
												arCameraResult[5,4,9+bYCounter]:=sCamera_To_Plc.iS03Result[i];	
											ELSIF i =15 THEN
												arCameraResult[5,4,bYCounter]:=sCamera_To_Plc.iS03Result[i];
											ELSIF i =16 THEN
												arCameraResult[5,4,6+bYCounter]:=sCamera_To_Plc.iS03Result[i];
											END_IF	
									END_IF
									IF i =16 THEN
										station.iStepAuto:=160;
									END_IF	
								END_FOR	
							END_IF
					END_IF
			END_IF	
			
		160://Y循环+1
			bYCounter :=bYCounter +1 ;
			station.iStepAuto:=180;
			
		180://判断循环次数是否已到
			IF   bYCounter<=3 THEN
				station.iStepAuto:=110;
			ELSE
				station.iStepAuto:=190; 
			END_IF
		190:///X轴拍照流程完成
				 tsModuleProcess[bXCounter+1].xProcessCompleted:=TRUE;
				 tsModuleProcess[bXCounter+1].xQDataCompleted:=TRUE;
					station.iStepAuto:=200; 
		200://Y轴回拍照位置1
				fbYAxisMove.xMoveAuto[2]:=TRUE;
				IF  fbYAxisMove.xMoveInPos[2] THEN
					station.iStepAuto:=210;
				END_IF
		210://X循环 +1 
			bXCounter :=bXCounter +1;
			station.iStepAuto:=220;
		220://X循环判断
			IF   bXCounter<=2 THEN
				station.iStepAuto:=50;
			ELSE
				station.iStepAuto:=230; 
			END_IF	
		230://Z轴上升
				fbZAxisMove.xMoveAuto[1]:=TRUE;
			IF  fbXAxisMove.xMoveInPos[1] THEN
					station.iStepAuto:= 240;
			END_IF
		240://水平调整气缸松开
					fbHOZAdjustCyl_1.xAuto:=FALSE;
					fbHOZAdjustCyl_2.xAuto:=false;
					fbHOZAdjustCyl_3.xAuto:=false;
					fbHOZAdjustCyl_4.xAuto:=false;
					fbHOZAdjustCyl_5.xAuto:=false;
					fbHOZAdjustCyl_6.xAuto:=false;
					fbHOZAdjustCyl_7.xAuto:=false;
					fbHOZAdjustCyl_8.xAuto:=false;
				IF  fbHOZAdjustCyl_1.xHP_Delay AND 
					fbHOZAdjustCyl_2.xHP_Delay AND
					fbHOZAdjustCyl_3.xHP_Delay AND
					fbHOZAdjustCyl_4.xHP_Delay AND 
					fbHOZAdjustCyl_5.xHP_Delay AND 
					fbHOZAdjustCyl_6.xHP_Delay AND
					fbHOZAdjustCyl_7.xHP_Delay AND
					fbHOZAdjustCyl_8.xHP_Delay THEN
					station.iStepInit:=250;	
				END_IF
		250://XY轴回参考点
				fbXAxisMove.xMoveAuto[1]:=TRUE;
				fbYAxisMove.xMoveAuto[1]:=TRUE;
			IF	fbxAxisMove.xMoveInPos[1] AND 
				fbYAxisMove.xMoveInPos[1] THEN
					station.iStepAuto:= 260;
			END_IF
		260:////Restore_after_Estop_Process4 数据传输流程
			IF  station.xSingleRunning OR fbMachine[1].xTryRun THEN
					station.iStepAuto :=999;
			ELSIF tsModuleProcess[4].xProcessNotStarted AND NOT  tsModuleProcess[4].xProcessStarted THEN
					station.iStepAuto :=270; (*process not started*)
			ELSIF  tsModuleProcess[4].xProcessStarted AND NOT  tsModuleProcess[4].xProcessCompleted THEN
				 station.iStepAuto := 275;(*process started*)
			ELSIF  tsModuleProcess[4].xProcessCompleted AND NOT tsModuleProcess[4].xQDataCompleted  THEN
					station.iStepAuto :=350;(*process completed*)
			ELSIF tsModuleProcess[4].xQDataCompleted THEN
					station.iStepAuto :=360;(*Qdata completed *)
			ELSE
					station.iStepAuto :=270; 
			END_IF		
		270://		
				tsModuleProcess[4].xProcessNotStarted:=TRUE;
				station.iStepAuto :=275; 
				
		275://储存结果
			tsModuleProcess[4].xProcessStarted:=TRUE;
			FOR i:=1 TO 5 BY 1 DO
				MEMCPY(ADR(arProcessDataStation[i].stProcessData.arCameraResult),ADR(arCameraResult[i,1,1]),
				SIZEOF(arProcessDataStation[i].stProcessData.arCameraResult));
			END_FOR
			station.iStepAuto:=280;
		280://汇总结果【4】
				FOR i:=1 TO 4 BY 1 DO
					FOR j :=1 TO 12 BY 1 DO 
						IF bCounter = 2 OR bCounter = 3 OR bEndCounter =1 THEN
							IF arProcessDataStation[4].stProcessData.arCameraResult[i,j]<> 1 THEN
								arProcessDataStation[4].stProduct.xLidChecking_NOK:=TRUE;
								arProcessDataStation[4].stProduct.xLidChecking_OK:=FALSE;
								EXIT;
							ELSIF   i=4 AND j =12 THEN
								arProcessDataStation[4].stProduct.xLidChecking_NOK:=FALSE;
								arProcessDataStation[4].stProduct.xLidChecking_OK:=TRUE;
								
							END_IF
						END_IF
					END_FOR
				END_FOR
				station.iStepAuto:=290;
		290://汇总结果【5】	
				FOR i:=1 TO 4 BY 1 DO
					FOR j :=1 TO 12 BY 1 DO 
						IF bCounter = 3  OR bEndCounter =2 THEN
							IF arProcessDataStation[5].stProcessData.arCameraResult[i,j]<>1 THEN
								arProcessDataStation[5].stProduct.xLidChecking_NOK:=TRUE;
								arProcessDataStation[5].stProduct.xLidChecking_OK:=FALSE;
								EXIT;
							ELSIF  i=4 AND j =12 THEN
								arProcessDataStation[5].stProduct.xLidChecking_NOK:=FALSE;
								arProcessDataStation[5].stProduct.xLidChecking_OK:=TRUE; 
							END_IF
						END_IF
					END_FOR
				END_FOR
				tsModuleProcess[4].xProcessCompleted:=TRUE;
				station.iStepAuto:=350;
		350://数据load
			IF  bCounter =1 OR bCounter =2 OR bCounter=3 THEN
				MEMCPY(ADR(arMainlineFixtureData[arCurFixtureNumStation[5]]),ADR(arProcessDataStation[1]),SIZEOF(arProcessDataStation[1]));
				MEMCPY(ADR(arMainlineFixtureData[arCurFixtureNumStation[6]]),ADR(arProcessDataStation[2]),SIZEOF(arProcessDataStation[2]));
			END_IF
			IF bCounter =2 OR bCounter =3 OR bEndCounter =1 THEN
				MEMCPY(ADR(arMainlineFixtureData[arCurFixtureNumStation[7]]),ADR(arProcessDataStation[3]),SIZEOF(arProcessDataStation[3]));
				MEMCPY(ADR(arMainlineFixtureData[arCurFixtureNumStation[8]]),ADR(arProcessDataStation[4]),SIZEOF(arProcessDataStation[4]));
			END_IF
			IF bCounter =3 OR bEndCounter =2 THEN
				MEMCPY(ADR(arMainlineFixtureData[arCurFixtureNumStation[9]]),ADR(arProcessDataStation[5]),SIZEOF(arProcessDataStation[5]));
			END_IF
				station.iStepAuto:= 360;
 		360://循环计数
			tsModuleProcess[4].xQDataCompleted:=TRUE;
			IF   bEndCounter =0 THEN
				bCounter:=bCounter +1;
			ELSIF  bCounter =0 THEN
				bEndCounter := bEndCounter +1;
			END_IF
			station.iStepAuto:=370;
			
		370://循环统计
			IF  bCounter >3 THEN
				bCounter :=3;
			END_IF
			station.iStepAuto:=999;
		
	////产品流程结束
	999://----Single Run Finish----
		arManualNOKHmiButton[3]:=FALSE;
		station.iStepAuto :=0;
		IF NOT station.xSingleContinuousRun THEN
			station.xSingleRunFlag:=FALSE;
		END_IF
		
		station.xCycleEnable:=FALSE;	
		station.xDone:=TRUE;
		station.xRunningOffProhibit := FALSE ;//运行中信号Off禁止
	ELSE
		;	
END_CASE



END_IF
END_ACTION

ACTION FlowInit:
IF NOT station.xIniting THEN
  station.iStepInit:=0;    
ELSE
//--------------------------------------------初始化步序----------------------------------
CASE station.iStepInit OF	
 0://  
  	IF station.xIniting THEN	
  	  station.iStepInit:=10;	
  	END_IF	
10://复位数据
	FOR i:=2 TO 17 BY 1 DO
		fbCamera[i].xlInit:=TRUE;
	END_FOR
	station.iStepInit :=20;
	 
20://伺服上电
  	 fbXAxisMove.xPowerInit := TRUE ;
	 fbYAxisMove.xPowerInit := TRUE ;
	 fbZAxisMove.xPowerInit := TRUE ;
	IF fbXAxisMove.xPowerOn AND   fbYAxisMove.xPowerOn AND  fbZAxisMove.xPowerOn THEN 
    	station.iStepInit:=30;	
	END_IF
30://Z轴伺服上升
		fbZAxisMove.xMoveAuto[1]:=TRUE;
		IF fbZAxisMove.xMoveInPos[1]   THEN
			station.iStepInit:=40;	
		END_IF
40://XY轴回参考位置
		fbXAxisMove.xMoveAuto[1]:=TRUE;
		fbYAxisMove.xMoveAuto[1]:=TRUE;
		IF fbXAxisMove.xMoveInPos[1]  AND   fbYAxisMove.xMoveInPos[1]  THEN
			station.iStepInit:=50;	
		END_IF
50://水平调整气缸回原位
		
		fbHOZAdjustCyl_1.xinit:=TRUE;
        fbHOZAdjustCyl_2.xinit:=true;
        fbHOZAdjustCyl_3.xinit:=true;
        fbHOZAdjustCyl_4.xinit:=true;
        fbHOZAdjustCyl_5.xinit:=true;
        fbHOZAdjustCyl_6.xinit:=true;
        fbHOZAdjustCyl_7.xinit:=true;
        fbHOZAdjustCyl_8.xinit:=TRUE;
	IF  fbHOZAdjustCyl_1.xHP_Delay AND 
		fbHOZAdjustCyl_2.xHP_Delay AND
		fbHOZAdjustCyl_3.xHP_Delay AND
		fbHOZAdjustCyl_4.xHP_Delay AND 
		fbHOZAdjustCyl_5.xHP_Delay AND 
		fbHOZAdjustCyl_6.xHP_Delay AND
		fbHOZAdjustCyl_7.xHP_Delay AND
		fbHOZAdjustCyl_8.xHP_Delay THEN
		station.iStepInit:=60;	
	END_IF

60://
	station.iStepInit:=100;

100://	
    station.iStepInit:=999;	
999://初始化完成	
	station.iStepInit:=0;
	station.xInitDone:=TRUE;  
END_CASE
END_IF
END_ACTION

ACTION General:
(******************清除过程记录**********************)
CASE bClearProcessStep OF
	0:	
		IF	 S08_MainLine.xClearProcessStatus THEN
			FOR i:=1 TO gc_ModuleProNo BY 1 DO
				MEMSET(ADR(tsModuleProcess[i]),0,SIZEOF(tsModuleProcess[i]));
			END_FOR
			bClearProcessStep:=10;
		END_IF
	10:
		xClearModuleProcessDone:=TRUE;
		bClearProcessStep:=20;
	20:
		IF NOT S08_MainLine.xClearProcessStatus THEN
			xClearModuleProcessDone:=FALSE;
			bClearProcessStep:=30;
		END_IF
	30:  
			bClearProcessStep:=0;
	
END_CASE

(*******************拍照结果放到HMI中**********************)
MEMCPY(ADR(arCameraResultHmi),ADR(arCameraResult),SIZEOF(arCameraResultHmi));
END_ACTION

ACTION ILC:

//---------------------------------------------------工站可执行-------------------------------------------------------
station.xCanRun :=TRUE ;

//---------------------------------------------------气缸动作条件-------------------------------------------
fbHOZAdjustCyl_1.xOffILC	:=	TRUE	;
fbHOZAdjustCyl_1.xOnILC	:=	TRUE	;
fbHOZAdjustCyl_2.xOffILC	:=	TRUE	;
fbHOZAdjustCyl_2.xOnILC	:=	TRUE	;
fbHOZAdjustCyl_3.xOffILC	:=	TRUE	;
fbHOZAdjustCyl_3.xOnILC	:=	TRUE	;
fbHOZAdjustCyl_4.xOffILC	:=	TRUE	;
fbHOZAdjustCyl_4.xOnILC	:=	TRUE	;
fbHOZAdjustCyl_5.xOffILC	:=	TRUE	;
fbHOZAdjustCyl_5.xOnILC	:=	TRUE	;
fbHOZAdjustCyl_6.xOffILC	:=	TRUE	;
fbHOZAdjustCyl_6.xOnILC	:=	TRUE	;
fbHOZAdjustCyl_7.xOffILC	:=	TRUE	;
fbHOZAdjustCyl_7.xOnILC	:=	TRUE	;
fbHOZAdjustCyl_8.xOffILC	:=	TRUE	;
fbHOZAdjustCyl_8.xOnILC	:=	TRUE	;


//---------------------------------------------------伺服动作条件-------------------------------------------

fbXAxisMove.xRunILC := 		
fbXAxisMove.xMoveILC[1] :=		
fbxAxisMove.xMoveILC[2] :=		
fbxAxisMove.xMoveILC[3] :=		
fbxAxisMove.xMoveILC[4] :=		
fbxAxisMove.xMoveILC[5] := 		fbZAxisMove.xMoveInPos[1] OR fbZAxisMove.xMoveInPos[2] ;
fbYAxisMove.xRunILC := 		
fbYAxisMove.xMoveILC[1] :=		
fbYAxisMove.xMoveILC[2] :=		
fbYAxisMove.xMoveILC[3] :=		
fbYAxisMove.xMoveILC[4] :=		
fbYAxisMove.xMoveILC[5] := 		fbZAxisMove.xMoveInPos[1] OR fbZAxisMove.xMoveInPos[2] ;
fbZAxisMove.xRunILC := 		
fbZAxisMove.xMoveILC[1] :=		
fbZAxisMove.xMoveILC[2] :=		
fbZAxisMove.xMoveILC[3] :=		
fbZAxisMove.xMoveILC[4] :=		
fbZAxisMove.xMoveILC[5] := 		TRUE;
END_ACTION

ACTION TipAuto:

//------------------------------------------------AutoTip Cylinder--------------------------------
station.adwAutoTip[1].00	:=	fbHOZAdjustCyl_1.xAutoTip	;
station.adwAutoTip[1].01	:=	fbHOZAdjustCyl_2.xAutoTip	;
station.adwAutoTip[1].02	:=	fbHOZAdjustCyl_3.xAutoTip	;
station.adwAutoTip[1].03	:=	fbHOZAdjustCyl_4.xAutoTip	;
station.adwAutoTip[1].04	:=	fbHOZAdjustCyl_5.xAutoTip	;
station.adwAutoTip[1].05	:=	fbHOZAdjustCyl_6.xAutoTip	;
station.adwAutoTip[1].06	:=	fbHOZAdjustCyl_7.xAutoTip	;
station.adwAutoTip[1].07	:=	fbHOZAdjustCyl_8.xAutoTip	;

//------------------------------------------------AutoTip Servo--------------------------------
//**************************************
FOR i:= 1 TO 5 BY 1 DO 
	IF fbXAxisMove.xMoveAuto[i] THEN
		fbXAxisMove.iPosNumber := i ;
	END_IF
	IF fbYAxisMove.xMoveAuto[i] THEN
		fbYAxisMove.iPosNumber := i ;
	END_IF
	IF fbZAxisMove.xMoveAuto[i] THEN
		fbZAxisMove.iPosNumber := i ;
	END_IF
	
END_FOR


IF  fbMachine[1].xAutoMode AND NOT fbMachine[1].xRunning  THEN
	  arTonDelay[01](IN:=True , PT:=T#1S , Q=> , ET=> );
else
	  arTonDelay[01](IN:=false);
END_IF
IF arTonDelay[1].Q  THEN 
		IF fbXAxisMove.iPosNumber=1 AND NOT fbXAxisMove.xMoveInPos[1] THEN station.adwAutoTip[1].10:=TRUE; END_IF//轴伺服自动时位置不在位置1	
		IF fbXAxisMove.iPosNumber=2 AND NOT fbXAxisMove.xMoveInPos[2] THEN station.adwAutoTip[1].11:=TRUE; END_IF//轴伺服自动时位置不在位置2	
		IF fbXAxisMove.iPosNumber=3 AND NOT fbXAxisMove.xMoveInPos[3] THEN station.adwAutoTip[1].12:=TRUE; END_IF//轴伺服自动时位置不在位置3	
		IF fbXAxisMove.iPosNumber=4 AND NOT fbXAxisMove.xMoveInPos[4] THEN station.adwAutoTip[1].13:=TRUE; END_IF//轴伺服自动时位置不在位置4	
		IF fbXAxisMove.iPosNumber=5 AND NOT fbXAxisMove.xMoveInPos[5] THEN station.adwAutoTip[1].14:=TRUE; END_IF//轴伺服自动时位置不在位置5	
		
		
		IF fbYAxisMove.iPosNumber=1 AND NOT fbYAxisMove.xMoveInPos[1] THEN station.adwAutoTip[1].15:=TRUE; END_IF//轴伺服自动时位置不在位置1	
		IF fbYAxisMove.iPosNumber=2 AND NOT fbYAxisMove.xMoveInPos[2] THEN station.adwAutoTip[1].16:=TRUE; END_IF//轴伺服自动时位置不在位置2	
		IF fbYAxisMove.iPosNumber=3 AND NOT fbYAxisMove.xMoveInPos[3] THEN station.adwAutoTip[1].17:=TRUE; END_IF//轴伺服自动时位置不在位置3	
		IF fbYAxisMove.iPosNumber=4 AND NOT fbYAxisMove.xMoveInPos[4] THEN station.adwAutoTip[1].18:=TRUE; END_IF//轴伺服自动时位置不在位置4	
		IF fbYAxisMove.iPosNumber=5 AND NOT fbYAxisMove.xMoveInPos[5] THEN station.adwAutoTip[1].19:=TRUE; END_IF//轴伺服自动时位置不在位置5	
		
		IF fbZAxisMove.iPosNumber=1 AND NOT fbZAxisMove.xMoveInPos[1] THEN station.adwAutoTip[1].20:=TRUE; END_IF//轴伺服自动时位置不在位置1	
		IF fbZAxisMove.iPosNumber=2 AND NOT fbZAxisMove.xMoveInPos[2] THEN station.adwAutoTip[1].21:=TRUE; END_IF//轴伺服自动时位置不在位置2	
		IF fbZAxisMove.iPosNumber=3 AND NOT fbZAxisMove.xMoveInPos[3] THEN station.adwAutoTip[1].22:=TRUE; END_IF//轴伺服自动时位置不在位置3	
		IF fbZAxisMove.iPosNumber=4 AND NOT fbZAxisMove.xMoveInPos[4] THEN station.adwAutoTip[1].23:=TRUE; END_IF//轴伺服自动时位置不在位置4	
		IF fbZAxisMove.iPosNumber=5 AND NOT fbZAxisMove.xMoveInPos[5] THEN station.adwAutoTip[1].24:=TRUE; END_IF//轴伺服自动时位置不在位置5			
END_IF
END_ACTION

ACTION TipManual:
//--------------------------------------------ManualTip------------------------------------------------------

//-------------------------------------------气缸提示---------------------------------------------------------




/////////////////////////////////////////////////////////////////////////////////////////////////////////////////
END_ACTION

ACTION Z_Output:
(**************************气缸输出********************************)
QxS03HOZAdjustCyl_1WP	:=	fbHOZAdjustCyl_1.xWP_Valve	;
QxS03HOZAdjustCyl_1HP	:=	fbHOZAdjustCyl_1.xHP_Valve	;
QxS03HOZAdjustCyl_2WP	:=	fbHOZAdjustCyl_2.xWP_Valve	;
QxS03HOZAdjustCyl_2HP	:=	fbHOZAdjustCyl_2.xHP_Valve	;
QxS03HOZAdjustCyl_3WP	:=	fbHOZAdjustCyl_3.xWP_Valve	;
QxS03HOZAdjustCyl_3HP	:=	fbHOZAdjustCyl_3.xHP_Valve	;
QxS03HOZAdjustCyl_4WP	:=	fbHOZAdjustCyl_4.xWP_Valve	;
QxS03HOZAdjustCyl_4HP	:=	fbHOZAdjustCyl_4.xHP_Valve	;
QxS03HOZAdjustCyl_5WP	:=	fbHOZAdjustCyl_5.xWP_Valve	;
QxS03HOZAdjustCyl_5HP	:=	fbHOZAdjustCyl_5.xHP_Valve	;
QxS03HOZAdjustCyl_6WP	:=	fbHOZAdjustCyl_6.xWP_Valve	;
QxS03HOZAdjustCyl_6HP	:=	fbHOZAdjustCyl_6.xHP_Valve	;
QxS03HOZAdjustCyl_7WP	:=	fbHOZAdjustCyl_7.xWP_Valve	;
QxS03HOZAdjustCyl_7HP	:=	fbHOZAdjustCyl_7.xHP_Valve	;
QxS03HOZAdjustCyl_8WP	:=	fbHOZAdjustCyl_8.xWP_Valve	;
QxS03HOZAdjustCyl_8HP	:=	fbHOZAdjustCyl_8.xHP_Valve	;
END_ACTION

END_PROGRAM

(* stored: Version 1.1.0.1, ProductVersion 3.1.4024.9
   POU S03_LidChecking: Id {77a9bd2b-7da1-438e-b565-cc8f27eee63e}, SpecialFunc None
   Action A_Input: Id {b6530cbb-368d-4144-89d4-ce2dff9991be}
   Action Alarm: Id {a083e1a6-5ad3-41b2-bcc4-4b4a15412287}
   Action Delay: Id {c3be7dc0-30a5-4d49-9e30-1bde31c71398}
   Action FlowAuto: Id {07295eb9-26b2-4b33-8e3f-eeb1088e4f36}
   Action FlowInit: Id {50953df4-ff4f-4c49-ba0d-1f4d4bb7faa6}
   Action General: Id {173921ed-8271-4b09-9710-611e1cae1f98}
   Action ILC: Id {b7f5a1ac-a880-4cb0-819a-4a4442b7778e}
   Action TipAuto: Id {22541172-1c77-494b-a7c8-1c43ec47b24b}
   Action TipManual: Id {dbaa108a-e0d4-4501-933e-e36048ea6f81}
   Action Z_Output: Id {110cf067-dbbf-4e5d-8ee0-386447e50660} *)
